(* IEC 61131-3 sources: volt/packages/volt-lsp-iec/test-corpus/pro2193/Device/Plc Logic/Application/09 Misc/Library Manager/BrinkEdgePcLogging (part 2) *)

(* ---- PRODUCTIONCOUNTERSPLCDATATYPESCONFIG.dut ---- *)
TYPE PRODUCTIONCOUNTERSPLCDATATYPESCONFIG : ARRAY [0..GVL_Dashboard.MaxNumberOfCavitiesRobot] OF CavityPlcDataTypes;
END_TYPE

(* ---- RESULT.dut ---- *)
TYPE RESULT :
(
	SUCCESS := 0,
	NOELEMENTS := 1,
	QUEUEFULL := 3,
	ALREADYLOCKED := 4
);
END_TYPE

(* ---- SENDDATATYPE.dut ---- *)
TYPE SENDDATATYPE :
(
	INIT := 1,
	KEEPALIVE := 2,
	NORMALRECORD := 3,
	STRINGRECORD := 4
);
END_TYPE

(* ---- STRINGLOGCACHE.dut ---- *)
TYPE STRINGLOGCACHE : ARRAY [1..QueuesInCache] OF StringLogQueue;
END_TYPE

(* ---- STRINGLOGRECORD.dut ---- *)
TYPE STRINGLOGRECORD :
STRUCT
	PLCDATATYPE : PlcDataType;
	DATATYPE : DataType;
	PLCUTCTIME : ULINT;
	VALUE : STRING(255);
END_STRUCT
END_TYPE

(* ---- STRINGLOGRECORDARRAY.dut ---- *)
TYPE STRINGLOGRECORDARRAY : ARRAY [1..GVL_Dashboard.StringLogQueueLength] OF StringLogRecord;
END_TYPE

(* ---- TCPCLIENTSTATE.dut ---- *)
TYPE TCPCLIENTSTATE :
(
	CONNECTINIT := 1,
	CONNECTING := 2,
	CONNECTED := 10,
	SENDING := 11,
	DISCONNECTED := -1,
	DISCONNECTING := -2
);
END_TYPE

(* ---- TCPWRITERESULT.dut ---- *)
TYPE TCPWRITERESULT :
(
	SUCCESS := 1,
	NOTYETCOMPLETED := 2,
	ERRORWHILESENDING := 3,
	DATATOOLONG := 4,
	ALREADYBUSY := 5,
	TOOMANYWRITESPERCYCLE := 6
);
END_TYPE

(* ---- XUVACUUMSPLCDATATYPESCONFIG.dut ---- *)
TYPE XUVACUUMSPLCDATATYPESCONFIG : ARRAY [1..2, 1..32] OF PlcDataType;
END_TYPE

(* ---- DASHBOARDMONITORINGPARAMETERS.gvl ---- *)
VAR_GLOBAL
	MAXINTSMONITORED : UINT := 60;
	MAXBOOLSMONITORED : UINT := 25;
	MAXREALSMONITORED : UINT := 70;
	MAXSTRINGSMONITORED : UINT := 15;
END_VAR

(* ---- DASHBOARDPARAMETERS.gvl ---- *)
VAR_GLOBAL
	MAXBUFFERTIMEONNOCONNECTION : TIME := TIME#1s500ms;
	NUMBEROFDEBUGLOGRECORDS : BYTE (1..100) := 100;
	TCPCONNECTTIMEOUT : TIME := TIME#2s500ms;
	MAXTCPRECONNECTDELAY : TIME := TIME#30s0ms;
	QUEUESINCACHE : BYTE (1..12) := 8;
END_VAR

(* ---- GVL_DASHBOARD.gvl ---- *)
VAR_GLOBAL
	MAXNUMBEROFCAVITIESROBOT : __UXINT := 64;
	SIZELOGRECORD : __UXINT := XSIZEOF(LogRecord);
	LOGQUEUELENGTH : BYTE := 110;
	SIZELOGQUEUE : __UXINT := (XSIZEOF(LogRecord) * LogQueueLength);
	SIZESTRINGLOGRECORD : __UXINT := XSIZEOF(StringLogRecord);
	STRINGLOGQUEUELENGTH : BYTE := 10;
	SIZESTRINGLOGQUEUE : __UXINT := (XSIZEOF(StringLogRecord) * StringLogQueueLength);
	TCPSENDARRAYLENGTH : UDINT := 2732;
END_VAR

(* ---- IADDLOG.itf ---- *)
INTERFACE IADDLOG
END_INTERFACE

METHOD ADDLOGBOOL : BOOL
VAR_INPUT
	PLCDATATYPE : PlcDataType;
	VALUE : BOOL;
END_VAR
END_METHOD

METHOD ADDLOGLINT : BOOL
VAR_INPUT
	PLCDATATYPE : PlcDataType;
	VALUE : LINT;
END_VAR
END_METHOD

METHOD ADDLOGLREAL : BOOL
VAR_INPUT
	PLCDATATYPE : PlcDataType;
	VALUE : LREAL;
END_VAR
END_METHOD

METHOD ADDLOGSTRING : BOOL
VAR_INPUT
	PLCDATATYPE : PlcDataType;
	VALUE : STRING(255);
END_VAR
END_METHOD

METHOD ADDLOGULINT : BOOL
VAR_INPUT
	PLCDATATYPE : PlcDataType;
	VALUE : ULINT;
END_VAR
END_METHOD

(* ---- GENERATELABELADJUSTMENTSPLCDATATYPESCONFIG.pou ---- *)
FUNCTION GENERATELABELADJUSTMENTSPLCDATATYPESCONFIG
VAR_INPUT
	LABELADJUSTMENTSCONFIG : REFERENCE TO LabelAdjustmentsPlcDataTypesConfig;
END_VAR
END_FUNCTION

(* ---- GENERATEMOULDCONTROLCAVITYPLCDATATYPESCONFIG.pou ---- *)
FUNCTION GENERATEMOULDCONTROLCAVITYPLCDATATYPESCONFIG
VAR_INPUT
	MOULDCONTROLCONFIG : REFERENCE TO MouldControlCavityPlcDataTypesConfig;
END_VAR
END_FUNCTION

(* ---- GENERATEMVACUUMSPLCDATATYPESCONFIG.pou ---- *)
FUNCTION GENERATEMVACUUMSPLCDATATYPESCONFIG
VAR_INPUT
	MVACUUMSCONFIG : REFERENCE TO MVacuumsPlcDataTypesConfig;
END_VAR
END_FUNCTION

(* ---- GENERATEPRODUCTIONCOUNTERSPLCDATATYPESCONFIG.pou ---- *)
FUNCTION GENERATEPRODUCTIONCOUNTERSPLCDATATYPESCONFIG
VAR_INPUT
	COUNTERSCONFIG : REFERENCE TO ProductionCountersPlcDataTypesConfig;
END_VAR
END_FUNCTION

(* ---- GENERATEXUVACUUMSPLCDATATYPESCONFIG.pou ---- *)
FUNCTION GENERATEXUVACUUMSPLCDATATYPESCONFIG
VAR_INPUT
	XUVACUUMSCONFIG : REFERENCE TO XuVacuumsPlcDataTypesConfig;
END_VAR
END_FUNCTION

(* ---- LOGWARNING.pou ---- *)
FUNCTION LOGWARNING
VAR_INPUT
	MESSAGE : STRING(80);
END_VAR
END_FUNCTION

(* ---- RELEASELOCK.pou ---- *)
FUNCTION RELEASELOCK : Result
VAR_IN_OUT
	LOCKVAR : DWORD;
END_VAR
END_FUNCTION

(* ---- TRYLOCK.pou ---- *)
FUNCTION TRYLOCK : BOOL
VAR_IN_OUT
	LOCKVAR : DWORD;
END_VAR
END_FUNCTION

(* ---- EDGEPCCLIENT.pou ---- *)
FUNCTION_BLOCK EDGEPCCLIENT
VAR_INPUT
	SERSERIALNO : STRING(10);
	IPV4ADDRESS : STRING(15) := '10.195.0.8';
	PORT : UINT := 48000;
	CONNECT : BOOL := TRUE;
	LOGCACHE : REFERENCE TO LogCache;
	STRINGLOGCACHE : REFERENCE TO StringLogCache;
	CONNSPEED : ConnectionSpeed := ConnectionSpeed.S100Mbps;
	CYCLEMS : BYTE := 4;
END_VAR
VAR
	LOGCACHEREFVALID : BOOL := FALSE;
	STRINGLOGCACHEREFVALID : BOOL := FALSE;
	TCPCLIENT : NBS.TCP_Client;
	IPADDRESS : NBS.IP_ADDR;
	TCPCLIENTACTIVE : BOOL := FALSE;
	TCPWRITE : NBS.TCP_Write;
	TCPREAD : NBS.TCP_Read;
	TCPREADBUFFER : ARRAY [1..256] OF BYTE;
	TCPREADBUFFERSIZE : __UXINT := XSIZEOF(tcpReadBuffer);
	STATE : TcpClientState := TcpClientState.Disconnected;
	CURRENTTIME : ULINT;
	RECONNECTTIMER : TON;
	RECONNECTDELAY : TIME := minReconnectInterval;
	CONNECTTIMER : TON;
	DEBUGMODE : BOOL := FALSE;
	DEBUGLOGS : ARRAY [1..DashboardParameters.NumberOfDebugLogRecords] OF DebugLogInfo;
	DEBUGLOGINDEX : USINT := 0;
	STATISTICS : ClientStatistics;
	KEEPALIVETIMER : TOF;
	AUTOCLOSETIMER : TOF;
	AUTOCLOSETIMERACTIVE : BOOL := FALSE;
	LONGDISCONNECTTIMER : TON;
	DISCONNECTEDSTATE : BOOL := FALSE;
	I : INT;
	SENDARR : ARRAY [1..GVL_Dashboard.TCPSendArrayLength] OF BYTE;
	SENDARRLOCK : DWORD;
	WRITESPERCYCLE : BYTE;
	MAXWRITESPERCYCLE : BYTE;
	NOTALLDATAWRITTEN : BOOL;
	TOTALSTART : ULINT;
	TOTALEND : ULINT;
	TOTALTIME : ULINT;
	MAXWRITETIME : ULINT;
	KEEPALIVEINTERVAL : TIME := TIME#250ms;
	AUTOCLOSEINTERVAL : TIME := TIME#5s0ms;
	MINRECONNECTINTERVAL : TIME := TIME#500ms;
	BOOLDATATYPE : DataType := DataType.boolean;
	LINTDATATYPE : DataType := DataType.integer;
	ULINTDATATYPE : DataType := DataType.ulinteger;
	LREALDATATYPE : DataType := DataType.float;
	BUSY : BOOL;
	CONNECTED : BOOL;
	CURRENTTIMEMS : ULINT;
	LONGDISCONNECTED : BOOL;
END_VAR
END_FUNCTION_BLOCK

METHOD CLOSECLIENTCONNECTION
END_METHOD

METHOD UPDATECURRENTTIME
END_METHOD

METHOD WRITEKEEPALIVE : BOOL
END_METHOD

METHOD WRITE : TcpWriteResult
VAR_INPUT
	PDATA : CAA.PVOID;
	DATALENGTH : CAA.SIZE;
	SENDDATATYPE : SendDataType;
END_VAR
END_METHOD

METHOD WRITEDEBUGLOG
VAR_INPUT
	DESCRIPTION : STRING(255);
END_VAR
END_METHOD

METHOD ONCONNECT : BOOL
END_METHOD

METHOD WRITEINITIAL : TcpWriteResult
END_METHOD

METHOD MONITORCONNECTINGCLIENT
END_METHOD

METHOD INCREASERECONNECTDELAY
END_METHOD

METHOD WRITELOGSTOCLIENT : BOOL
END_METHOD

METHOD ADDLOGBOOL : BOOL
VAR_INPUT
	PLCDATATYPE : PlcDataType;
	VALUE : BOOL;
END_VAR
END_METHOD

METHOD ADDLOG : BOOL
VAR_INPUT
	PLCDATATYPE : PlcDataType;
	DATATYPE : DataType;
	VALUE : NumberUnion;
END_VAR
END_METHOD

METHOD ADDLOGLREAL : BOOL
VAR_INPUT
	PLCDATATYPE : PlcDataType;
	VALUE : LREAL;
END_VAR
END_METHOD

METHOD ADDLOGULINT : BOOL
VAR_INPUT
	PLCDATATYPE : PlcDataType;
	VALUE : ULINT;
END_VAR
END_METHOD

METHOD ADDLOGLINT : BOOL
VAR_INPUT
	PLCDATATYPE : PlcDataType;
	VALUE : LINT;
END_VAR
END_METHOD

METHOD ADDLOGSTRING : BOOL
VAR_INPUT
	PLCDATATYPE : PlcDataType;
	VALUE : STRING(255);
END_VAR
END_METHOD

(* ---- LINTCHANGEDTRIGGER.pou ---- *)
FUNCTION_BLOCK LINTCHANGEDTRIGGER
VAR_INPUT
	INPUT : LINT;
	MAXDIFF : LINT;
END_VAR
VAR_OUTPUT
	Q : BOOL;
	DIFF : LINT;
END_VAR
VAR
	LASTINPUT : LINT;
END_VAR
END_FUNCTION_BLOCK

METHOD SETLASTINPUT
VAR_INPUT
	VALUE : LINT;
END_VAR
END_METHOD

(* ---- LOGQUEUE.pou ---- *)
FUNCTION_BLOCK LOGQUEUE
VAR_OUTPUT
	LOGQUEUE : LogRecordArray;
	FULL : BOOL := FALSE;
	EMPTY : BOOL := TRUE;
END_VAR
VAR
	LASTUSEDINDEX : DINT (0..GVL_Dashboard.LogQueueLength) := 0;
	LOCKVAR : DWORD;
	TOTALLOGSADDED : ULINT;
	COUNT : DINT;
END_VAR
END_FUNCTION_BLOCK

METHOD TRYADD : Result
VAR_INPUT
	PLCDATATYPE : PlcDataType;
	DATATYPE : DataType;
	PLCUTCTIME : ULINT;
	VALUE : NumberUnion;
END_VAR
END_METHOD

METHOD CLEAR : Result
END_METHOD

METHOD UNSAFECLEAR
END_METHOD

METHOD REQUESTLOCK : BOOL
END_METHOD

METHOD UNLOCK
END_METHOD

(* ---- LREALCHANGEDTRIGGER.pou ---- *)
FUNCTION_BLOCK LREALCHANGEDTRIGGER
VAR_INPUT
	INPUT : LREAL;
	MAXDIFF : LREAL;
END_VAR
VAR_OUTPUT
	Q : BOOL;
	DIFF : LREAL;
END_VAR
VAR
	LASTINPUT : LREAL;
END_VAR
END_FUNCTION_BLOCK

METHOD SETLASTINPUT
VAR_INPUT
	VALUE : LREAL;
END_VAR
END_METHOD

(* ---- MONITORANYINT.pou ---- *)
FUNCTION_BLOCK MONITORANYINT EXTENDS MonitorBase
VAR
	REFINPUT : POINTER TO AnyNumber;
	INPUTTYPE : __SYSTEM.TYPE_CLASS;
	INPUTISSIGNED : BOOL;
	INPUTISULINT : BOOL;
	CURRENTINPUT : AnyNumber := STRUCT(ULINTval := 0);
	OLDVALUE : AnyNumber := STRUCT(ULINTval := 0);
	DIFF : UDINT (0..1000);
	TIMEOUT : TIME;
	CHANGEDTIMER : Standard.TON;
	SENDZEROFIRST : BOOL;
	FORCESEND : BOOL := FALSE;
	FORCESENDZERO : BOOL := FALSE;
	LINTCHANGED : LINTChangedTrigger;
	ULINTCHANGED : ULINTChangedTrigger;
END_VAR
END_FUNCTION_BLOCK

METHOD INITIALIZE
VAR_INPUT
	PLCDATATYPE : PlcDataType;
	VALUE : __SYSTEM.AnyType;
	DIFF : UDINT (0..1000);
	TIMEOUT : TIME := TIME#10s0ms;
	SENDONEDGEPCCONNECT : BOOL := FALSE;
	SENDONINTERVAL : TIME := TIME#0ms;
	SENDZEROFIRST : BOOL := FALSE;
END_VAR
END_METHOD

METHOD RESETCHANGEDTRIGGERTOOLDVALUE
END_METHOD

METHOD LOGCURRENTINPUT : BOOL
END_METHOD

METHOD INITIALIZEINTERNAL
VAR_INPUT
	PLCDATATYPE : PlcDataType;
	VALUE : __SYSTEM.AnyType;
	DIFF : UDINT (0..1000);
	TIMEOUT : TIME := TIME#10s0ms;
	SENDONEDGEPCCONNECT : BOOL := FALSE;
	SENDONINTERVAL : TIME := TIME#0ms;
	SENDZEROFIRST : BOOL := FALSE;
END_VAR
END_METHOD

(* ---- MONITORANYREAL.pou ---- *)
FUNCTION_BLOCK MONITORANYREAL EXTENDS MonitorBase
VAR
	P4 : POINTER TO REAL;
	P8 : POINTER TO LREAL;
	SIZE : DINT;
	DIFF : REAL := 0.1;
	TRIGGER : LREALChangedTrigger;
	CURRENTVALUE : LREAL;
	OLDVALUE : LREAL;
END_VAR
END_FUNCTION_BLOCK

METHOD INITIALIZE
VAR_INPUT
	PLCDATATYPE : PlcDataType;
	VALUE : __SYSTEM.AnyType;
	DIFF : REAL := 0.1;
	SENDONEDGEPCCONNECT : BOOL := FALSE;
	SENDONINTERVAL : TIME := TIME#0ms;
END_VAR
END_METHOD

METHOD INITIALIZEINTERNAL
VAR_INPUT
	PLCDATATYPE : PlcDataType;
	VALUE : __SYSTEM.AnyType;
	DIFF : REAL := 0.1;
	SENDONEDGEPCCONNECT : BOOL := FALSE;
	SENDONINTERVAL : TIME := TIME#0ms;
END_VAR
END_METHOD

(* ---- MONITORBASE.pou ---- *)
FUNCTION_BLOCK MONITORBASE
VAR
	LOGGINGFB : IAddLog;
	PLCDATATYPE : PlcDataType;
	INTERVAL : Standard.TON;
	SENDONEDGEPCCONNECT : BOOL;
	SENDONINTERVAL : TIME;
	TRIGGEREDGEPCCONNECT : Standard.R_TRIG;
	EDGEPCCONNECTTRIGGER : BOOL;
END_VAR
END_FUNCTION_BLOCK

METHOD SETCLIENT
VAR_INPUT
	LOGGINGFB : IAddLog;
END_VAR
END_METHOD

(* ---- MONITORBOOLEAN.pou ---- *)
FUNCTION_BLOCK MONITORBOOLEAN EXTENDS MonitorBase
VAR
	REFINPUT : REFERENCE TO BOOL;
	OLDVALUE : BOOL;
END_VAR
END_FUNCTION_BLOCK

METHOD INITIALIZE
VAR_INPUT
	PLCDATATYPE : PlcDataType;
	REFINPUT : REFERENCE TO BOOL;
	SENDONEDGEPCCONNECT : BOOL := FALSE;
	SENDONINTERVAL : TIME := TIME#0ms;
END_VAR
END_METHOD

(* ---- MONITORINGSERVICE.pou ---- *)
FUNCTION_BLOCK MONITORINGSERVICE
VAR_INPUT
	EDGEPCCLIENT : IAddLog;
END_VAR
VAR
	REGISTERINGLOCK : DWORD := 0;
	I : UINT;
	MONITORINT : ARRAY [1..DashboardMonitoringParameters.MaxIntsMonitored] OF MonitorAnyInt;
	MONITORBOOL : ARRAY [1..DashboardMonitoringParameters.MaxBoolsMonitored] OF MonitorBoolean;
	MONITORREAL : ARRAY [1..DashboardMonitoringParameters.MaxRealsMonitored] OF MonitorAnyReal;
	MONITORSTRING : ARRAY [1..DashboardMonitoringParameters.MaxStringsMonitored] OF MonitorString;
	ACTUALINTSMONITORED : UINT := 0;
	ACTUALBOOLSMONITORED : UINT := 0;
	ACTUALREALSMONITORED : UINT := 0;
	ACTUALSTRINGSMONITORED : UINT := 0;
	INTMONITORSEXTRANEEDED : UINT := 0;
	BOOLMONITORSEXTRANEEDED : UINT := 0;
	REALMONITORSEXTRANEEDED : UINT := 0;
	STRINGMONITORSEXTRANEEDED : UINT := 0;
END_VAR
END_FUNCTION_BLOCK

METHOD UNREGISTERALL
END_METHOD

METHOD REGISTERBOOL : BOOL
VAR_INPUT
	PLCDATATYPE : PlcDataType;
	REFINPUT : REFERENCE TO BOOL;
	SENDONEDGEPCCONNECT : BOOL := FALSE;
	SENDONINTERVAL : TIME := TIME#0ms;
END_VAR
END_METHOD

METHOD INITIALIZE : BOOL
VAR_INPUT
	FORCE : BOOL := FALSE;
END_VAR
END_METHOD

METHOD REGISTERINT : BOOL
VAR_INPUT
	PLCDATATYPE : PlcDataType;
	VALUE : __SYSTEM.AnyType;
	DIFF : UDINT (0..1000);
	TIMEOUT : TIME := TIME#10s0ms;
	SENDONEDGEPCCONNECT : BOOL := FALSE;
	SENDONINTERVAL : TIME := TIME#0ms;
	SENDZEROFIRST : BOOL := FALSE;
END_VAR
END_METHOD

METHOD REGISTERREAL : BOOL
VAR_INPUT
	PLCDATATYPE : PlcDataType;
	VALUE : __SYSTEM.AnyType;
	DIFF : REAL := 0.1;
	SENDONEDGEPCCONNECT : BOOL := FALSE;
	SENDONINTERVAL : TIME := TIME#0ms;
END_VAR
END_METHOD

METHOD REGISTERSTRING : BOOL
VAR_INPUT
	PLCDATATYPE : PlcDataType;
	REFINPUT : Stu.CharBufferPtr;
	SENDONEDGEPCCONNECT : BOOL := FALSE;
	SENDONINTERVAL : TIME := TIME#0ms;
END_VAR
END_METHOD

(* ---- MONITORSTRING.pou ---- *)
FUNCTION_BLOCK MONITORSTRING EXTENDS MonitorBase
VAR
	REFINPUT : Stu.CharBufferPtr;
	REFINPUTLENGTH : DINT;
	CURRENTVALUE : STRING(255);
	OLDVALUE : STRING(255);
	COMPARERESULT : INT;
END_VAR
END_FUNCTION_BLOCK

METHOD INITIALIZE
VAR_INPUT
	PLCDATATYPE : PlcDataType;
	REFINPUT : Stu.CharBufferPtr;
	SENDONEDGEPCCONNECT : BOOL := FALSE;
	SENDONINTERVAL : TIME := TIME#0ms;
END_VAR
END_METHOD

(* ---- STRINGLOGQUEUE.pou ---- *)
FUNCTION_BLOCK STRINGLOGQUEUE
VAR_OUTPUT
	LOGQUEUE : StringLogRecordArray;
	FULL : BOOL := FALSE;
	EMPTY : BOOL := TRUE;
END_VAR
VAR
	LASTUSEDINDEX : DINT (0..GVL_Dashboard.StringLogQueueLength) := 0;
	LOCKVAR : DWORD;
	TOTALLOGSADDED : ULINT;
	STRINGDATATYPE : DataType := DataType.text;
	COUNT : DINT;
END_VAR
END_FUNCTION_BLOCK

METHOD TRYADD : Result
VAR_INPUT
	PLCDATATYPE : PlcDataType;
	PLCUTCTIME : ULINT;
	VALUE : STRING(255);
END_VAR
END_METHOD

METHOD CLEAR : Result
END_METHOD

METHOD UNSAFECLEAR
END_METHOD

METHOD REQUESTLOCK : BOOL
END_METHOD

METHOD UNLOCK
END_METHOD

(* ---- ULINTCHANGEDTRIGGER.pou ---- *)
FUNCTION_BLOCK ULINTCHANGEDTRIGGER
VAR_INPUT
	INPUT : ULINT;
	MAXDIFF : ULINT;
END_VAR
VAR_OUTPUT
	Q : BOOL;
	DIFF : ULINT;
END_VAR
VAR
	LASTINPUT : ULINT;
END_VAR
END_FUNCTION_BLOCK

METHOD SETLASTINPUT
VAR_INPUT
	VALUE : ULINT;
END_VAR
END_METHOD
